INTERFACE I_SerialControlledDevice

METHOD StartSend : BOOL
VAR_INPUT
END_VAR
END_METHOD

METHOD StopSend : BOOL
VAR_INPUT
END_VAR
END_METHOD

END_INTERFACE

(* stored: Version 1.1.0.1, ProductVersion 3.1.4024.9
   Itf I_SerialControlledDevice: Id {65f13558-6a7f-4359-8026-07cf4695500c}
   Method StartSend: Id {c4217205-e4d8-4cf7-b323-d74f4f9ceec2}
   Method StopSend: Id {a996e6f4-dbcd-479b-85d0-ccfe2ec25da2} *)
